// TIA Portal V18 export
// export: Created 2026-03-12T16:04:34.6564057Z, ExportSetting WithDefaults, DisplayName Totally Integrated Automation Portal, DisplayVersion V18 Update 5, DisplayName TIA Portal Openness, DisplayVersion V18 Update 5, DisplayName TIA Portal Version Control Interface, DisplayVersion V18, DisplayName SINAMICS Startdrive Advanced, DisplayVersion V18, DisplayName SINAMICS Startdrive G130, G150, S120, S150, SINAMICS MV, S210, DisplayVersion V18, DisplayName SINAMICS Startdrive G110M, G120, G120C, G120D, G120P, G115D, DisplayVersion V18, DisplayName STEP 7 Professional, DisplayVersion V18 Update 5, DisplayName STEP 7 Safety, DisplayVersion V18, DisplayName WinCC Professional, DisplayVersion V18 Update 5
FUNCTION_BLOCK "FB INVERSOR SIEMENS"   // FB20, LAD
{ S7_Optimized_Access := 'TRUE' }
VERSION : 0.1
// stored: AutoNumber true, IsIECCheckEnabled false, IsRetainMemResEnabled false, MemoryReserve 100, SetENOAutomatically false, UDAEnableTagReadback false
   VAR_INPUT
      RPM_min_Driver : Int;
      RPM_Max_Driver : Int;
      Setpoint_Velocidade : Int;
   END_VAR
   VAR_OUTPUT
      Telegram_Out_Velocidade : Int;
   END_VAR
   VAR_TEMP
      Aux_Velocidade : Real;
   END_VAR
BEGIN

REGION Network 1: Controle Velocidade
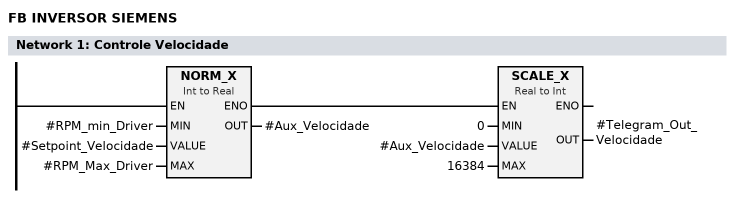
   RUNG wire#powerrail
      { S7_Templates := "[SrcType := Int, DestType := Real]" } Normalize(min := #RPM_min_Driver, value := #Setpoint_Velocidade, max := #RPM_Max_Driver, out => #Aux_Velocidade)
      { S7_Templates := "[SrcType := Real, DestType := Int]" } Scale(min := 0, value := #Aux_Velocidade, max := 16384, out => #Telegram_Out_Velocidade)
   END_RUNG
   // the same network as SCL:
   #Aux_Velocidade := NORM_X(MIN := #RPM_min_Driver, VALUE := #Setpoint_Velocidade, MAX := #RPM_Max_Driver);
   #Telegram_Out_Velocidade := SCALE_X(MIN := 0, VALUE := #Aux_Velocidade, MAX := 16384);
END_REGION
END_FUNCTION_BLOCK
